PROGRAM TestStationSensors
VAR
	(* These timers are used to imitate the moving time in the visualization*)
	t1: TIME := TIME#500MS;
	TON_0: TON;
	TON_1: TON;
	
END_VAR
VAR // added by the converter: edge detectors and wires of the graphical bodies
    _w1, _w2 : BOOL;
END_VAR

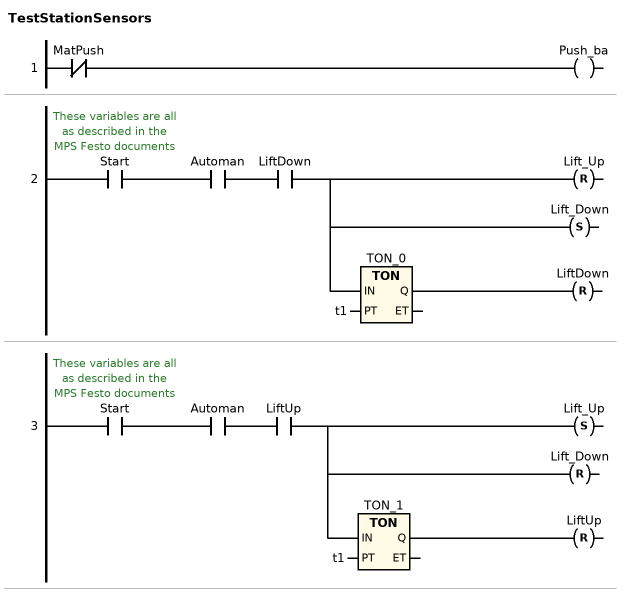
// NETWORK 1
Push_ba := NOT MatPush;

// NETWORK 2
//   Start: These variables are all as described in the MPS Festo documents
_w1 := Start AND Automan AND LiftDown;
Lift_Up R= _w1;
Lift_Down S= _w1;
TON_0(IN := _w1, PT := t1); // TON
LiftDown R= TON_0.Q;

// NETWORK 3
//   Start: These variables are all as described in the MPS Festo documents
_w2 := Start AND Automan AND LiftUp;
Lift_Up S= _w2;
Lift_Down R= _w2;
TON_1(IN := _w2, PT := t1); // TON
LiftUp R= TON_1.Q;

END_PROGRAM

(* stored: Version 1.1.0.1, ProductVersion 3.1.4018.5
   POU TestStationSensors: Id {787d885e-9c7e-4065-9515-e03aee25a41b}, SpecialFunc None *)
